// TIA Portal V17 export
// export: Created 2024-09-02T12:50:37.3880681Z, ExportSetting WithDefaults, DisplayName Totally Integrated Automation Portal, DisplayVersion V17, DisplayName TIA Portal Openness, DisplayVersion V17, DisplayName TIA Portal Version Control Interface, DisplayVersion V17, DisplayName STEP 7 Professional, DisplayVersion V17, DisplayName STEP 7 Safety, DisplayVersion V17, DisplayName WinCC Professional, DisplayVersion V17
TYPE "Proces_r"
// stored: IsFailsafeCompliant false
   STRUCT
      "Finished OK" : Bool;
      "Finished NOK" : Bool;
      Repeated : Bool;
      Reserve_1 : Bool;
      Reserve_2 : Bool;
      Reserve_3 : Bool;
      "OK Operator decision" : Bool;
      "NOK Operator decision" : Bool;
   END_STRUCT;
END_TYPE
